{attribute 'qualified_only'}
VAR_GLOBAL CONSTANT
    Good                                 : DINT := 16#00000000; // The operation succeeded.
    Uncertain                            : DINT := 16#40000000; // The operation was uncertain.
    Bad                                  : DINT := 16#80000000; // The operation failed.
    BadUnexpectedError                   : DINT := 16#80010000; // An unexpected error occurred.
    BadInternalError                     : DINT := 16#80020000; // An internal error occurred as a result of a programming or configuration error.
    BadOutOfMemory                       : DINT := 16#80030000; // Not enough memory to complete the operation.
    BadResourceUnavailable               : DINT := 16#80040000; // An operating system resource is not available.
    BadCommunicationError                : DINT := 16#80050000; // A low level communication error occurred.
    BadEncodingError                     : DINT := 16#80060000; // Encoding halted because of invalid data in the objects being serialized.
    BadDecodingError                     : DINT := 16#80070000; // Decoding halted because of invalid data in the stream.
    BadEncodingLimitsExceeded            : DINT := 16#80080000; // The message encoding/decoding limits imposed by the stack have been exceeded.
    BadRequestTooLarge                   : DINT := 16#80B80000; // The request message size exceeds limits set by the server.
    BadResponseTooLarge                  : DINT := 16#80B90000; // The response message size exceeds limits set by the client or server.
    BadUnknownResponse                   : DINT := 16#80090000; // An unrecognized response was received from the server.
    BadTimeout                           : DINT := 16#800A0000; // The operation timed out.
    BadServiceUnsupported                : DINT := 16#800B0000; // The server does not support the requested service.
    BadShutdown                          : DINT := 16#800C0000; // The operation was cancelled because the application is shutting down.
    BadServerNotConnected                : DINT := 16#800D0000; // The operation could not complete because the client is not connected to the server.
    BadServerHalted                      : DINT := 16#800E0000; // The server has stopped and cannot process any requests.
    BadNothingToDo                       : DINT := 16#800F0000; // No processing could be done because there was nothing to do.
    BadTooManyOperations                 : DINT := 16#80100000; // The request could not be processed because it specified too many operations.
    BadTooManyMonitoredItems             : DINT := 16#80DB0000; // The request could not be processed because there are too many monitored items in the subscription.
    BadDataTypeIdUnknown                 : DINT := 16#80110000; // The extension object cannot be (de)serialized because the data type id is not recognized.
    BadCertificateInvalid                : DINT := 16#80120000; // The certificate provided as a parameter is not valid.
    BadSecurityChecksFailed              : DINT := 16#80130000; // An error occurred verifying security.
    BadCertificatePolicyCheckFailed      : DINT := 16#81140000; // The certificate does not meet the requirements of the security policy.
    BadCertificateTimeInvalid            : DINT := 16#80140000; // The certificate has expired or is not yet valid.
    BadCertificateIssuerTimeInvalid      : DINT := 16#80150000; // An issuer certificate has expired or is not yet valid.
    BadCertificateHostNameInvalid        : DINT := 16#80160000; // The HostName used to connect to a server does not match a HostName in the certificate.
    BadCertificateUriInvalid             : DINT := 16#80170000; // The URI specified in the ApplicationDescription does not match the URI in the certificate.
    BadCertificateUseNotAllowed          : DINT := 16#80180000; // The certificate may not be used for the requested operation.
    BadCertificateIssuerUseNotAllowed    : DINT := 16#80190000; // The issuer certificate may not be used for the requested operation.
    BadCertificateUntrusted              : DINT := 16#801A0000; // The certificate is not trusted.
    BadCertificateRevocationUnknown      : DINT := 16#801B0000; // It was not possible to determine if the certificate has been revoked.
    BadCertificateIssuerRevocationUnknown: DINT := 16#801C0000; // It was not possible to determine if the issuer certificate has been revoked.
    BadCertificateRevoked                : DINT := 16#801D0000; // The certificate has been revoked.
    BadCertificateIssuerRevoked          : DINT := 16#801E0000; // The issuer certificate has been revoked.
    BadCertificateChainIncomplete        : DINT := 16#810D0000; // The certificate chain is incomplete.
    BadUserAccessDenied                  : DINT := 16#801F0000; // User does not have permission to perform the requested operation.
    BadIdentityTokenInvalid              : DINT := 16#80200000; // The user identity token is not valid.
    BadIdentityTokenRejected             : DINT := 16#80210000; // The user identity token is valid but the server has rejected it.
    BadSecureChannelIdInvalid            : DINT := 16#80220000; // The specified secure channel is no longer valid.
    BadInvalidTimestamp                  : DINT := 16#80230000; // The timestamp is outside the range allowed by the server.
    BadNonceInvalid                      : DINT := 16#80240000; // The nonce does appear to be not a random value or it is not the correct length.
    BadSessionIdInvalid                  : DINT := 16#80250000; // The session id is not valid.
    BadSessionClosed                     : DINT := 16#80260000; // The session was closed by the client.
    BadSessionNotActivated               : DINT := 16#80270000; // The session cannot be used because ActivateSession has not been called.
    BadSubscriptionIdInvalid             : DINT := 16#80280000; // The subscription id is not valid.
    BadRequestHeaderInvalid              : DINT := 16#802A0000; // The header for the request is missing or invalid.
    BadTimestampsToReturnInvalid         : DINT := 16#802B0000; // The timestamps to return parameter is invalid.
    BadRequestCancelledByClient          : DINT := 16#802C0000; // The request was cancelled by the client.
    BadTooManyArguments                  : DINT := 16#80E50000; // Too many arguments were provided.
    BadLicenseExpired                    : DINT := 16#810E0000; // The server requires a license to operate in general or to perform a service or operation, but existing license is expired.
    BadLicenseLimitsExceeded             : DINT := 16#810F0000; // The server has limits on number of allowed operations / objects, based on installed licenses, and these limits where exceeded.
    BadLicenseNotAvailable               : DINT := 16#81100000; // The server does not have a license which is required to operate in general or to perform a service or operation.
    BadServerTooBusy                     : DINT := 16#80EE0000; // The Server does not have the resources to process the request at this time.
    GoodPasswordChangeRequired           : DINT := 16#00EF0000; // The log-on for the user succeeded but the user is required to change the password.
    GoodSubscriptionTransferred          : DINT := 16#002D0000; // The subscription was transferred to another session.
    GoodCompletesAsynchronously          : DINT := 16#002E0000; // The processing will complete asynchronously.
    GoodOverload                         : DINT := 16#002F0000; // Sampling has slowed down due to resource limitations.
    GoodClamped                          : DINT := 16#00300000; // The value written was accepted but was clamped.
    BadNoCommunication                   : DINT := 16#80310000; // Communication with the data source is defined, but not established, and there is no last known value available.
    BadWaitingForInitialData             : DINT := 16#80320000; // Waiting for the server to obtain values from the underlying data source.
    BadNodeIdInvalid                     : DINT := 16#80330000; // The syntax the node id is not valid or refers to a node that is not valid for the operation.
    BadNodeIdUnknown                     : DINT := 16#80340000; // The node id refers to a node that does not exist in the server address space.
    BadAttributeIdInvalid                : DINT := 16#80350000; // The attribute is not supported for the specified Node.
    BadIndexRangeInvalid                 : DINT := 16#80360000; // The syntax of the index range parameter is invalid.
    BadIndexRangeNoData                  : DINT := 16#80370000; // No data exists within the range of indexes specified.
    BadIndexRangeDataMismatch            : DINT := 16#80EA0000; // The written data does not match the IndexRange specified.
    BadDataEncodingInvalid               : DINT := 16#80380000; // The data encoding is invalid.
    BadDataEncodingUnsupported           : DINT := 16#80390000; // The server does not support the requested data encoding for the node.
    BadNotReadable                       : DINT := 16#803A0000; // The access level does not allow reading or subscribing to the Node.
    BadNotWritable                       : DINT := 16#803B0000; // The access level does not allow writing to the Node.
    BadOutOfRange                        : DINT := 16#803C0000; // The value was out of range.
    BadNotSupported                      : DINT := 16#803D0000; // The requested operation is not supported.
    BadNotFound                          : DINT := 16#803E0000; // A requested item was not found or a search operation ended without success.
    BadObjectDeleted                     : DINT := 16#803F0000; // The object cannot be used because it has been deleted.
    BadNotImplemented                    : DINT := 16#80400000; // Requested operation is not implemented.
    BadMonitoringModeInvalid             : DINT := 16#80410000; // The monitoring mode is invalid.
    BadMonitoredItemIdInvalid            : DINT := 16#80420000; // The monitoring item id does not refer to a valid monitored item.
    BadMonitoredItemFilterInvalid        : DINT := 16#80430000; // The monitored item filter parameter is not valid.
    BadMonitoredItemFilterUnsupported    : DINT := 16#80440000; // The server does not support the requested monitored item filter.
    BadFilterNotAllowed                  : DINT := 16#80450000; // A monitoring filter cannot be used in combination with the attribute specified.
    BadStructureMissing                  : DINT := 16#80460000; // A mandatory structured parameter was missing or null.
    BadEventFilterInvalid                : DINT := 16#80470000; // The event filter is not valid.
    BadContentFilterInvalid              : DINT := 16#80480000; // The content filter is not valid.
    BadFilterOperatorInvalid             : DINT := 16#80C10000; // An unrecognized operator was provided in a filter.
    BadFilterOperatorUnsupported         : DINT := 16#80C20000; // A valid operator was provided, but the server does not provide support for this filter operator.
    BadFilterOperandCountMismatch        : DINT := 16#80C30000; // The number of operands provided for the filter operator was less then expected for the operand provided.
    BadFilterOperandInvalid              : DINT := 16#80490000; // The operand used in a content filter is not valid.
    BadFilterElementInvalid              : DINT := 16#80C40000; // The referenced element is not a valid element in the content filter.
    BadFilterLiteralInvalid              : DINT := 16#80C50000; // The referenced literal is not a valid value.
    BadContinuationPointInvalid          : DINT := 16#804A0000; // The continuation point provide is longer valid.
    BadNoContinuationPoints              : DINT := 16#804B0000; // The operation could not be processed because all continuation points have been allocated.
    BadReferenceTypeIdInvalid            : DINT := 16#804C0000; // The reference type id does not refer to a valid reference type node.
    BadBrowseDirectionInvalid            : DINT := 16#804D0000; // The browse direction is not valid.
    BadNodeNotInView                     : DINT := 16#804E0000; // The node is not part of the view.
    BadNumericOverflow                   : DINT := 16#81120000; // The number was not accepted because of a numeric overflow.
    BadLocaleNotSupported                : DINT := 16#80ED0000; // The locale in the requested write operation is not supported.
    BadNoValue                           : DINT := 16#80F00000; // The variable has no default value and no initial value.
    BadServerUriInvalid                  : DINT := 16#804F0000; // The ServerUri is not a valid URI.
    BadServerNameMissing                 : DINT := 16#80500000; // No ServerName was specified.
    BadDiscoveryUrlMissing               : DINT := 16#80510000; // No DiscoveryUrl was specified.
    BadSemaphoreFileMissing              : DINT := 16#80520000; // The semaphore file specified by the client is not valid.
    BadRequestTypeInvalid                : DINT := 16#80530000; // The security token request type is not valid.
    BadSecurityModeRejected              : DINT := 16#80540000; // The security mode does not meet the requirements set by the server.
    BadSecurityPolicyRejected            : DINT := 16#80550000; // The security policy does not meet the requirements set by the server.
    BadTooManySessions                   : DINT := 16#80560000; // The server has reached its maximum number of sessions.
    BadUserSignatureInvalid              : DINT := 16#80570000; // The user token signature is missing or invalid.
    BadApplicationSignatureInvalid       : DINT := 16#80580000; // The signature generated with the client certificate is missing or invalid.
    BadNoValidCertificates               : DINT := 16#80590000; // The client did not provide at least one software certificate that is valid and meets the profile requirements for the server.
    BadIdentityChangeNotSupported        : DINT := 16#80C60000; // The server does not support changing the user identity assigned to the session.
    BadRequestCancelledByRequest         : DINT := 16#805A0000; // The request was cancelled by the client with the Cancel service.
    BadParentNodeIdInvalid               : DINT := 16#805B0000; // The parent node id does not to refer to a valid node.
    BadReferenceNotAllowed               : DINT := 16#805C0000; // The reference could not be created because it violates constraints imposed by the data model.
    BadNodeIdRejected                    : DINT := 16#805D0000; // The requested node id was reject because it was either invalid or server does not allow node ids to be specified by the client.
    BadNodeIdExists                      : DINT := 16#805E0000; // The requested node id is already used by another node.
    BadNodeClassInvalid                  : DINT := 16#805F0000; // The node class is not valid.
    BadBrowseNameInvalid                 : DINT := 16#80600000; // The browse name is invalid.
    BadBrowseNameDuplicated              : DINT := 16#80610000; // The browse name is not unique among nodes that share the same relationship with the parent.
    BadNodeAttributesInvalid             : DINT := 16#80620000; // The node attributes are not valid for the node class.
    BadTypeDefinitionInvalid             : DINT := 16#80630000; // The type definition node id does not reference an appropriate type node.
    BadSourceNodeIdInvalid               : DINT := 16#80640000; // The source node id does not reference a valid node.
    BadTargetNodeIdInvalid               : DINT := 16#80650000; // The target node id does not reference a valid node.
    BadDuplicateReferenceNotAllowed      : DINT := 16#80660000; // The reference type between the nodes is already defined.
    BadInvalidSelfReference              : DINT := 16#80670000; // The server does not allow this type of self reference on this node.
    BadReferenceLocalOnly                : DINT := 16#80680000; // The reference type is not valid for a reference to a remote server.
    BadNoDeleteRights                    : DINT := 16#80690000; // The server will not allow the node to be deleted.
    UncertainReferenceNotDeleted         : DINT := 16#40BC0000; // The server was not able to delete all target references.
    BadServerIndexInvalid                : DINT := 16#806A0000; // The server index is not valid.
    BadViewIdUnknown                     : DINT := 16#806B0000; // The view id does not refer to a valid view node.
    BadViewTimestampInvalid              : DINT := 16#80C90000; // The view timestamp is not available or not supported.
    BadViewParameterMismatch             : DINT := 16#80CA0000; // The view parameters are not consistent with each other.
    BadViewVersionInvalid                : DINT := 16#80CB0000; // The view version is not available or not supported.
    UncertainNotAllNodesAvailable        : DINT := 16#40C00000; // The list of references may not be complete because the underlying system is not available.
    GoodResultsMayBeIncomplete           : DINT := 16#00BA0000; // The server should have followed a reference to a node in a remote server but did not. The result set may be incomplete.
    BadNotTypeDefinition                 : DINT := 16#80C80000; // The provided Nodeid was not a type definition nodeid.
    UncertainReferenceOutOfServer        : DINT := 16#406C0000; // One of the references to follow in the relative path references to a node in the address space in another server.
    BadTooManyMatches                    : DINT := 16#806D0000; // The requested operation has too many matches to return.
    BadQueryTooComplex                   : DINT := 16#806E0000; // The requested operation requires too many resources in the server.
    BadNoMatch                           : DINT := 16#806F0000; // The requested operation has no match to return.
    BadMaxAgeInvalid                     : DINT := 16#80700000; // The max age parameter is invalid.
    BadSecurityModeInsufficient          : DINT := 16#80E60000; // The operation is not permitted over the current secure channel.
    BadHistoryOperationInvalid           : DINT := 16#80710000; // The history details parameter is not valid.
    BadHistoryOperationUnsupported       : DINT := 16#80720000; // The server does not support the requested operation.
    BadInvalidTimestampArgument          : DINT := 16#80BD0000; // The defined timestamp to return was invalid.
    BadWriteNotSupported                 : DINT := 16#80730000; // The server does not support writing the combination of value, status and timestamps provided.
    BadTypeMismatch                      : DINT := 16#80740000; // The value supplied for the attribute is not of the same type as the attribute's value.
    BadMethodInvalid                     : DINT := 16#80750000; // The method id does not refer to a method for the specified object.
    BadArgumentsMissing                  : DINT := 16#80760000; // The client did not specify all of the input arguments for the method.
    BadNotExecutable                     : DINT := 16#81110000; // The executable attribute does not allow the execution of the method.
    BadTooManySubscriptions              : DINT := 16#80770000; // The server has reached its maximum number of subscriptions.
    BadTooManyPublishRequests            : DINT := 16#80780000; // The server has reached the maximum number of queued publish requests.
    BadNoSubscription                    : DINT := 16#80790000; // There is no subscription available for this session.
    BadSequenceNumberUnknown             : DINT := 16#807A0000; // The sequence number is unknown to the server.
    GoodRetransmissionQueueNotSupported  : DINT := 16#00DF0000; // The Server does not support retransmission queue and acknowledgement of sequence numbers is not available.
    BadMessageNotAvailable               : DINT := 16#807B0000; // The requested notification message is no longer available.
    BadInsufficientClientProfile         : DINT := 16#807C0000; // The client of the current session does not support one or more Profiles that are necessary for the subscription.
    BadStateNotActive                    : DINT := 16#80BF0000; // The sub-state machine is not currently active.
    BadAlreadyExists                     : DINT := 16#81150000; // An equivalent rule already exists.
    BadTcpServerTooBusy                  : DINT := 16#807D0000; // The server cannot process the request because it is too busy.
    BadTcpMessageTypeInvalid             : DINT := 16#807E0000; // The type of the message specified in the header invalid.
    BadTcpSecureChannelUnknown           : DINT := 16#807F0000; // The SecureChannelId and/or TokenId are not currently in use.
    BadTcpMessageTooLarge                : DINT := 16#80800000; // The size of the message chunk specified in the header is too large.
    BadTcpNotEnoughResources             : DINT := 16#80810000; // There are not enough resources to process the request.
    BadTcpInternalError                  : DINT := 16#80820000; // An internal error occurred.
    BadTcpEndpointUrlInvalid             : DINT := 16#80830000; // The server does not recognize the QueryString specified.
    BadRequestInterrupted                : DINT := 16#80840000; // The request could not be sent because of a network interruption.
    BadRequestTimeout                    : DINT := 16#80850000; // Timeout occurred while processing the request.
    BadSecureChannelClosed               : DINT := 16#80860000; // The secure channel has been closed.
    BadSecureChannelTokenUnknown         : DINT := 16#80870000; // The token has expired or is not recognized.
    BadSequenceNumberInvalid             : DINT := 16#80880000; // The sequence number is not valid.
    BadProtocolVersionUnsupported        : DINT := 16#80BE0000; // The applications do not have compatible protocol versions.
    BadConfigurationError                : DINT := 16#80890000; // There is a problem with the configuration that affects the usefulness of the value.
    BadNotConnected                      : DINT := 16#808A0000; // The variable should receive its value from another variable, but has never been configured to do so.
    BadDeviceFailure                     : DINT := 16#808B0000; // There has been a failure in the device/data source that generates the value that has affected the value.
    BadSensorFailure                     : DINT := 16#808C0000; // There has been a failure in the sensor from which the value is derived by the device/data source.
    BadOutOfService                      : DINT := 16#808D0000; // The source of the data is not operational.
    BadDeadbandFilterInvalid             : DINT := 16#808E0000; // The deadband filter is not valid.
    UncertainNoCommunicationLastUsableValue: DINT := 16#408F0000; // Communication to the data source has failed. The variable value is the last value that had a good quality.
    UncertainLastUsableValue             : DINT := 16#40900000; // Whatever was updating this value has stopped doing so.
    UncertainSubstituteValue             : DINT := 16#40910000; // The value is an operational value that was manually overwritten.
    UncertainInitialValue                : DINT := 16#40920000; // The value is an initial value for a variable that normally receives its value from another variable.
    UncertainSensorNotAccurate           : DINT := 16#40930000; // The value is at one of the sensor limits.
    UncertainEngineeringUnitsExceeded    : DINT := 16#40940000; // The value is outside of the range of values defined for this parameter.
    UncertainSubNormal                   : DINT := 16#40950000; // The data value is derived from multiple sources and has less than the required number of Good sources.
    GoodLocalOverride                    : DINT := 16#00960000; // The value has been overridden.
    GoodSubNormal                        : DINT := 16#00EB0000; // The value is derived from multiple sources and has the required number of Good sources, but less than the full number of Good sources.
    BadRefreshInProgress                 : DINT := 16#80970000; // This Condition refresh failed, a Condition refresh operation is already in progress.
    BadConditionAlreadyDisabled          : DINT := 16#80980000; // This condition has already been disabled.
    BadConditionAlreadyEnabled           : DINT := 16#80CC0000; // This condition has already been enabled.
    BadConditionDisabled                 : DINT := 16#80990000; // Property not available, this condition is disabled.
    BadEventIdUnknown                    : DINT := 16#809A0000; // The specified event id is not recognized.
    BadEventNotAcknowledgeable           : DINT := 16#80BB0000; // The event cannot be acknowledged.
    BadDialogNotActive                   : DINT := 16#80CD0000; // The dialog condition is not active.
    BadDialogResponseInvalid             : DINT := 16#80CE0000; // The response is not valid for the dialog.
    BadConditionBranchAlreadyAcked       : DINT := 16#80CF0000; // The condition branch has already been acknowledged.
    BadConditionBranchAlreadyConfirmed   : DINT := 16#80D00000; // The condition branch has already been confirmed.
    BadConditionAlreadyShelved           : DINT := 16#80D10000; // The condition has already been shelved.
    BadConditionNotShelved               : DINT := 16#80D20000; // The condition is not currently shelved.
    BadShelvingTimeOutOfRange            : DINT := 16#80D30000; // The shelving time not within an acceptable range.
    BadNoData                            : DINT := 16#809B0000; // No data exists for the requested time range or event filter.
    BadBoundNotFound                     : DINT := 16#80D70000; // No data found to provide upper or lower bound value.
    BadBoundNotSupported                 : DINT := 16#80D80000; // The server cannot retrieve a bound for the variable.
    BadDataLost                          : DINT := 16#809D0000; // Data is missing due to collection started/stopped/lost.
    BadDataUnavailable                   : DINT := 16#809E0000; // Expected data is unavailable for the requested time range due to an un-mounted volume, an off-line archive or tape, or similar reason for temporary unavailability.
    BadEntryExists                       : DINT := 16#809F0000; // The data or event was not successfully inserted because a matching entry exists.
    BadNoEntryExists                     : DINT := 16#80A00000; // The data or event was not successfully updated because no matching entry exists.
    BadTimestampNotSupported             : DINT := 16#80A10000; // The Client requested history using a TimestampsToReturn the Server does not support.
    GoodEntryInserted                    : DINT := 16#00A20000; // The data or event was successfully inserted into the historical database.
    GoodEntryReplaced                    : DINT := 16#00A30000; // The data or event field was successfully replaced in the historical database.
    UncertainDataSubNormal               : DINT := 16#40A40000; // The aggregate value is derived from multiple values and has less than the required number of Good values.
    GoodNoData                           : DINT := 16#00A50000; // No data exists for the requested time range or event filter.
    GoodMoreData                         : DINT := 16#00A60000; // More data is available in the time range beyond the number of values requested.
    BadAggregateListMismatch             : DINT := 16#80D40000; // The requested number of Aggregates does not match the requested number of NodeIds.
    BadAggregateNotSupported             : DINT := 16#80D50000; // The requested Aggregate is not support by the server.
    BadAggregateInvalidInputs            : DINT := 16#80D60000; // The aggregate value could not be derived due to invalid data inputs.
    BadAggregateConfigurationRejected    : DINT := 16#80DA0000; // The aggregate configuration is not valid for specified node.
    GoodDataIgnored                      : DINT := 16#00D90000; // The request specifies fields which are not valid for the EventType or cannot be saved by the historian.
    BadRequestNotAllowed                 : DINT := 16#80E40000; // The request was rejected by the server because it did not meet the criteria set by the server.
    BadRequestNotComplete                : DINT := 16#81130000; // The request has not been processed by the server yet.
    BadTransactionPending                : DINT := 16#80E80000; // The operation is not allowed because a transaction is in progress.
    BadTicketRequired                    : DINT := 16#811F0000; // The device identity needs a ticket before it can be accepted.
    BadTicketInvalid                     : DINT := 16#81200000; // The device identity needs a ticket before it can be accepted.
    BadLocked                            : DINT := 16#80E90000; // The requested operation is not allowed, because the Node is locked by a different application.
    BadRequiresLock                      : DINT := 16#80EC0000; // The requested operation is not allowed, because the Node is not locked by the application.
    GoodEdited                           : DINT := 16#00DC0000; // The value does not come from the real source and has been edited by the server.
    GoodPostActionFailed                 : DINT := 16#00DD0000; // There was an error in execution of these post-actions.
    UncertainDominantValueChanged        : DINT := 16#40DE0000; // The related EngineeringUnit has been changed but the Variable Value is still provided based on the previous unit.
    GoodDependentValueChanged            : DINT := 16#00E00000; // A dependent value has been changed but the change has not been applied to the device.
    BadDominantValueChanged              : DINT := 16#80E10000; // The related EngineeringUnit has been changed but this change has not been applied to the device. The Variable Value is still dependent on the previous unit but its status is currently Bad.
    UncertainDependentValueChanged       : DINT := 16#40E20000; // A dependent value has been changed but the change has not been applied to the device. The quality of the dominant variable is uncertain.
    BadDependentValueChanged             : DINT := 16#80E30000; // A dependent value has been changed but the change has not been applied to the device. The quality of the dominant variable is Bad.
    GoodEdited_DependentValueChanged     : DINT := 16#01160000; // It is delivered with a dominant Variable value when a dependent Variable has changed but the change has not been applied.
    GoodEdited_DominantValueChanged      : DINT := 16#01170000; // It is delivered with a dependent Variable value when a dominant Variable has changed but the change has not been applied.
    GoodEdited_DominantValueChanged_DependentValueChanged: DINT := 16#01180000; // It is delivered with a dependent Variable value when a dominant or dependent Variable has changed but change has not been applied.
    BadEdited_OutOfRange                 : DINT := 16#81190000; // It is delivered with a Variable value when Variable has changed but the value is not legal.
    BadInitialValue_OutOfRange           : DINT := 16#811A0000; // It is delivered with a Variable value when a source Variable has changed but the value is not legal.
    BadOutOfRange_DominantValueChanged   : DINT := 16#811B0000; // It is delivered with a dependent Variable value when a dominant Variable has changed and the value is not legal.
    BadEdited_OutOfRange_DominantValueChanged: DINT := 16#811C0000; // It is delivered with a dependent Variable value when a dominant Variable has changed, the value is not legal and the change has not been applied.
    BadOutOfRange_DominantValueChanged_DependentValueChanged: DINT := 16#811D0000; // It is delivered with a dependent Variable value when a dominant or dependent Variable has changed and the value is not legal.
    BadEdited_OutOfRange_DominantValueChanged_DependentValueChanged: DINT := 16#811E0000; // It is delivered with a dependent Variable value when a dominant or dependent Variable has changed, the value is not legal and the change has not been applied.
    GoodCommunicationEvent               : DINT := 16#00A70000; // The communication layer has raised an event.
    GoodShutdownEvent                    : DINT := 16#00A80000; // The system is shutting down.
    GoodCallAgain                        : DINT := 16#00A90000; // The operation is not finished and needs to be called again.
    GoodNonCriticalTimeout               : DINT := 16#00AA0000; // A non-critical timeout occurred.
    BadInvalidArgument                   : DINT := 16#80AB0000; // One or more arguments are invalid.
    BadConnectionRejected                : DINT := 16#80AC0000; // Could not establish a network connection to remote server.
    BadDisconnect                        : DINT := 16#80AD0000; // The server has disconnected from the client.
    BadConnectionClosed                  : DINT := 16#80AE0000; // The network connection has been closed.
    BadInvalidState                      : DINT := 16#80AF0000; // The operation cannot be completed because the object is closed, uninitialized or in some other invalid state.
    BadEndOfStream                       : DINT := 16#80B00000; // Cannot move beyond end of the stream.
    BadNoDataAvailable                   : DINT := 16#80B10000; // No data is currently available for reading from a non-blocking stream.
    BadWaitingForResponse                : DINT := 16#80B20000; // The asynchronous operation is waiting for a response.
    BadOperationAbandoned                : DINT := 16#80B30000; // The asynchronous operation was abandoned by the caller.
	BadExpectedStreamToBlock             : DINT := 16#80B40000; // The stream did not return all data requested (possibly because it is a non-blocking stream).
    BadWouldBlock                        : DINT := 16#80B50000; // Non blocking behaviour is required and the operation would block.
    BadSyntaxError                       : DINT := 16#80B60000; // A value had an invalid syntax.
    BadMaxConnectionsReached             : DINT := 16#80B70000; // The operation could not be finished because all available connections are in use.
    UncertainTransducerInManual          : DINT := 16#42080000; // The value may not be accurate because the transducer is in manual mode.
    UncertainSimulatedValue              : DINT := 16#42090000; // The value is simulated.
    UncertainSensorCalibration           : DINT := 16#420A0000; // The value may not be accurate due to a sensor calibration fault.
    UncertainConfigurationError          : DINT := 16#420F0000; // The value may not be accurate due to a configuration issue.
    GoodCascadeInitializationAcknowledged: DINT := 16#04010000; // The value source supports cascade handshaking and the value has been Initialized based on an initialization request from a cascade secondary.
    GoodCascadeInitializationRequest     : DINT := 16#04020000; // The value source supports cascade handshaking and is requesting initialization of a cascade primary.
    GoodCascadeNotInvited                : DINT := 16#04030000; // The value source supports cascade handshaking, however, the source’s current state does not allow for cascade.
    GoodCascadeNotSelected               : DINT := 16#04040000; // The value source supports cascade handshaking, however, the source has not selected the corresponding cascade primary for use.
    GoodFaultStateActive                 : DINT := 16#04070000; // There is a fault state condition active in the value source.
    GoodInitiateFaultState               : DINT := 16#04080000; // A fault state condition is being requested of the destination.
    GoodCascade                          : DINT := 16#04090000; // The value is accurate, and the signal source supports cascade handshaking.
    BadDataSetIdInvalid                  : DINT := 16#80E70000; // The DataSet specified for the DataSetWriter creation is invalid.
END_VAR

(* stored: Version 1.1.0.1
   GVL OpcUaStatusCodes: Id {880f46fb-fb2c-4f88-a7fb-cfa802e5aefb} *)
